# EPICS substitutions: CsHeaterApp/Db/Watlow_PM_Output_1.substitutions
file Watlow_PM_Output_1.template
{
pattern	{  s, ta,      ss, mod}
	{   , SE,  Watlow,   1}
}
